// TIA Portal V21 export
FUNCTION_BLOCK "FB104"   // FB104, LAD
TITLE = FB104
{ S7_Optimized_Access := 'FALSE' }
// MANUAL PID
// stored: AutoNumber false, SetENOAutomatically false
   VAR_INPUT
      Enable : Bool;
      SecPulse : Bool;
      AlwaysTrue : Bool;
      DigitalOrAnalog : Bool;   // 0: DIGITAL; 1: ANALOG
      InvertPIDSel : Bool;   // 0: NO; 1: YES
      ActValue : Real;
      SetValue : Real;
      SetPoint1 : Real := 5.0;
      SetPoint2 : Real := 10.0;
      SetPoint3 : Real := 15.0;
      SetPoint4 : Real := 20.0;
      SetPoint5 : Real := 25.0;
      SetPoint6 : Real := 30.0;
      SetPoint7 : Real := 35.0;
      SetPoint8 : Real := 40.0;
      SetPoint9 : Real := 45.0;
      SetPoint10 : Real := 50.0;
      SetRef1 : Real := 10.0;
      SetRef2 : Real := 20.0;
      SetRef3 : Real := 30.0;
      SetRef4 : Real := 40.0;
      SetRef5 : Real := 50.0;
      SetRef6 : Real := 60.0;
      SetRef7 : Real := 70.0;
      SetRef8 : Real := 80.0;
      SetRef9 : Real := 90.0;
      SetRef10 : Real := 100.0;
      OnTime1 : Int := 2;
      OnTime2 : Int := 2;
      OnTime3 : Int := 2;
      OnTime4 : Int := 2;
      OnTime5 : Int := 2;
      OnTime6 : Int := 2;
      OnTime7 : Int := 2;
      OnTime8 : Int := 2;
      OnTime9 : Int := 2;
      OnTime10 : Int := 2;
      OffTime1 : Int := 3;
      OffTime2 : Int := 3;
      OffTime3 : Int := 3;
      OffTime4 : Int := 3;
      OffTime5 : Int := 3;
      OffTime6 : Int := 3;
      OffTime7 : Int := 3;
      OffTime8 : Int := 3;
      OffTime9 : Int := 3;
      OffTime10 : Int := 3;
   END_VAR
   VAR_OUTPUT
      Valve : Bool;
      SetRef : Real;
   END_VAR
   VAR_IN_OUT
      ControlValue1 : Real;
      ControlValue2 : Real;
      ControlValue3 : Real;
      ControlValue4 : Real;
      ControlValue5 : Real;
      ControlValue6 : Real;
      ControlValue7 : Real;
      ControlValue8 : Real;
      ControlValue9 : Real;
      ControlValue10 : Real;
   END_VAR
   VAR
      OnOffDelay { S7_SetPoint := 'True'} : "FB102";
      OnTime : Int;
      OffTime : Int;
   END_VAR
   VAR_TEMP   // added for the SCL form of the ladder/FBD networks
      _w1 : Bool;
   END_VAR
BEGIN

REGION Network 1: Set Point Calculations
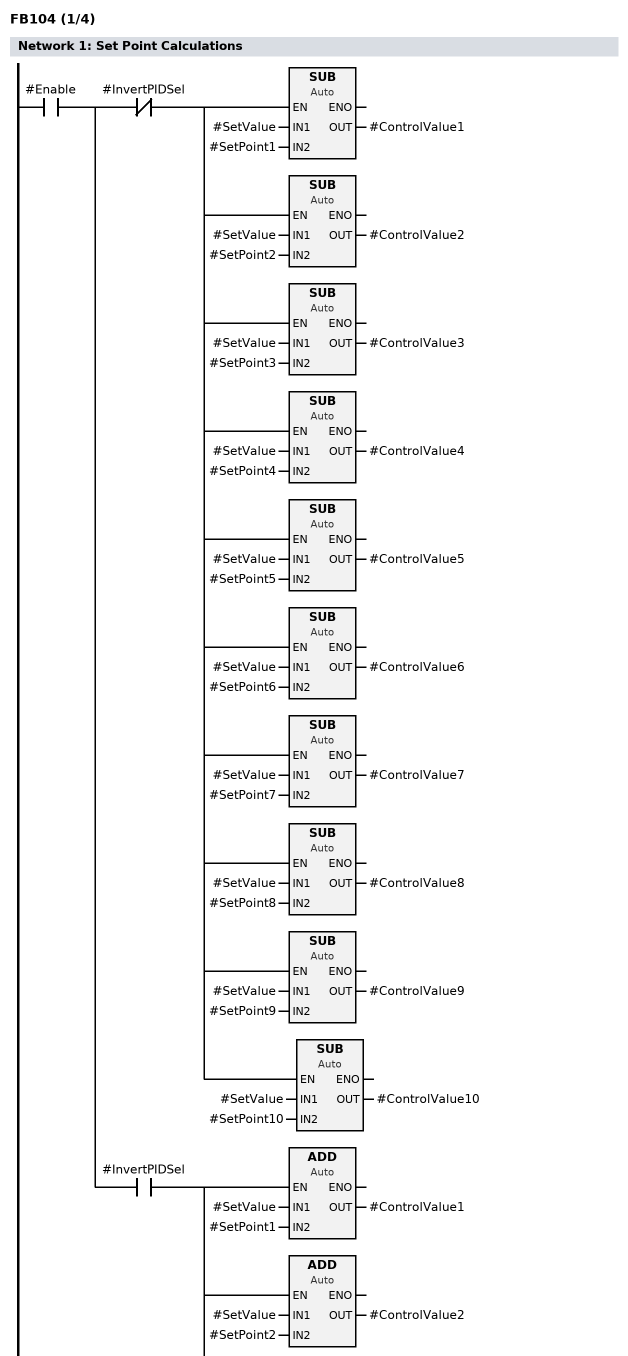
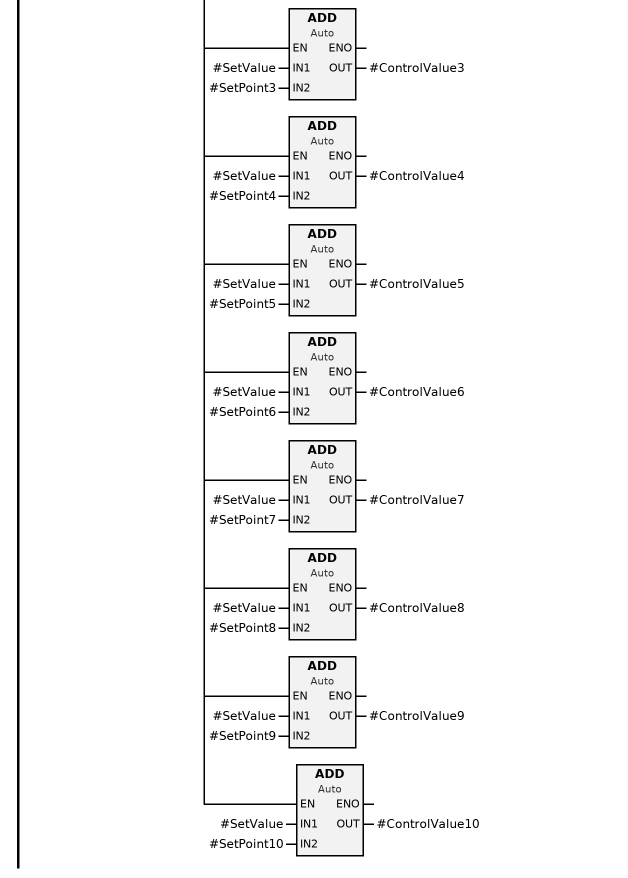
   RUNG wire#powerrail
      Contact( #Enable )
      wire#w1
      I_Contact( #InvertPIDSel )
      wire#w2
      Sub(in1 := #SetValue, in2 := #SetPoint1, out => #ControlValue1)
   END_RUNG
   RUNG wire#w2
      Sub(in1 := #SetValue, in2 := #SetPoint2, out => #ControlValue2)
   END_RUNG
   RUNG wire#w2
      Sub(in1 := #SetValue, in2 := #SetPoint3, out => #ControlValue3)
   END_RUNG
   RUNG wire#w2
      Sub(in1 := #SetValue, in2 := #SetPoint4, out => #ControlValue4)
   END_RUNG
   RUNG wire#w2
      Sub(in1 := #SetValue, in2 := #SetPoint5, out => #ControlValue5)
   END_RUNG
   RUNG wire#w2
      Sub(in1 := #SetValue, in2 := #SetPoint6, out => #ControlValue6)
   END_RUNG
   RUNG wire#w2
      Sub(in1 := #SetValue, in2 := #SetPoint7, out => #ControlValue7)
   END_RUNG
   RUNG wire#w2
      Sub(in1 := #SetValue, in2 := #SetPoint8, out => #ControlValue8)
   END_RUNG
   RUNG wire#w2
      Sub(in1 := #SetValue, in2 := #SetPoint9, out => #ControlValue9)
   END_RUNG
   RUNG wire#w2
      Sub(in1 := #SetValue, in2 := #SetPoint10, out => #ControlValue10)
   END_RUNG
   RUNG wire#w1
      Contact( #InvertPIDSel )
      wire#w3
      Add(in1 := #SetValue, in2 := #SetPoint1, out => #ControlValue1)
   END_RUNG
   RUNG wire#w3
      Add(in1 := #SetValue, in2 := #SetPoint2, out => #ControlValue2)
   END_RUNG
   RUNG wire#w3
      Add(in1 := #SetValue, in2 := #SetPoint3, out => #ControlValue3)
   END_RUNG
   RUNG wire#w3
      Add(in1 := #SetValue, in2 := #SetPoint4, out => #ControlValue4)
   END_RUNG
   RUNG wire#w3
      Add(in1 := #SetValue, in2 := #SetPoint5, out => #ControlValue5)
   END_RUNG
   RUNG wire#w3
      Add(in1 := #SetValue, in2 := #SetPoint6, out => #ControlValue6)
   END_RUNG
   RUNG wire#w3
      Add(in1 := #SetValue, in2 := #SetPoint7, out => #ControlValue7)
   END_RUNG
   RUNG wire#w3
      Add(in1 := #SetValue, in2 := #SetPoint8, out => #ControlValue8)
   END_RUNG
   RUNG wire#w3
      Add(in1 := #SetValue, in2 := #SetPoint9, out => #ControlValue9)
   END_RUNG
   RUNG wire#w3
      Add(in1 := #SetValue, in2 := #SetPoint10, out => #ControlValue10)
   END_RUNG
   // the same network as SCL:
   IF #Enable AND NOT #InvertPIDSel THEN
       #ControlValue1 := #SetValue - #SetPoint1;
       #ControlValue2 := #SetValue - #SetPoint2;
       #ControlValue3 := #SetValue - #SetPoint3;
       #ControlValue4 := #SetValue - #SetPoint4;
       #ControlValue5 := #SetValue - #SetPoint5;
       #ControlValue6 := #SetValue - #SetPoint6;
       #ControlValue7 := #SetValue - #SetPoint7;
       #ControlValue8 := #SetValue - #SetPoint8;
       #ControlValue9 := #SetValue - #SetPoint9;
       #ControlValue10 := #SetValue - #SetPoint10;
   END_IF;
   IF #Enable AND #InvertPIDSel THEN
       #ControlValue1 := #SetValue + #SetPoint1;
       #ControlValue2 := #SetValue + #SetPoint2;
       #ControlValue3 := #SetValue + #SetPoint3;
       #ControlValue4 := #SetValue + #SetPoint4;
       #ControlValue5 := #SetValue + #SetPoint5;
       #ControlValue6 := #SetValue + #SetPoint6;
       #ControlValue7 := #SetValue + #SetPoint7;
       #ControlValue8 := #SetValue + #SetPoint8;
       #ControlValue9 := #SetValue + #SetPoint9;
       #ControlValue10 := #SetValue + #SetPoint10;
   END_IF;
END_REGION

REGION Network 2: Set Reference for InvertPIDSel: NO
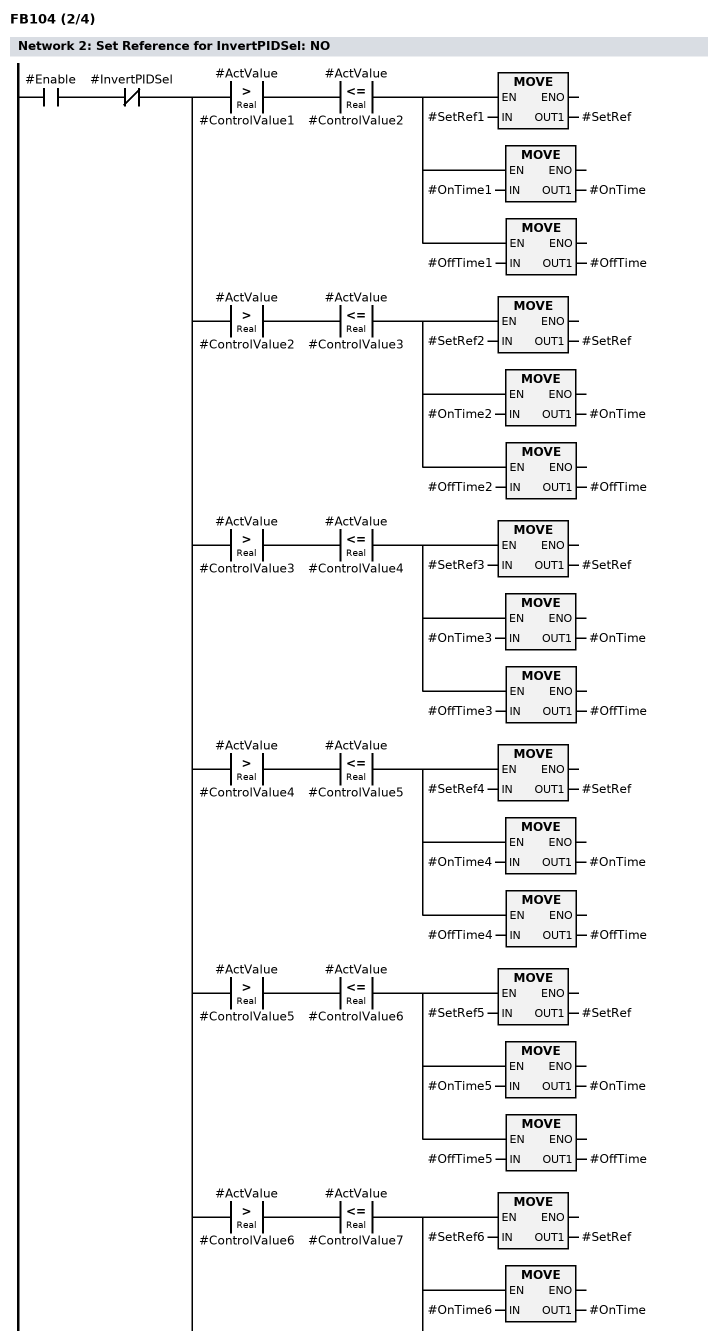
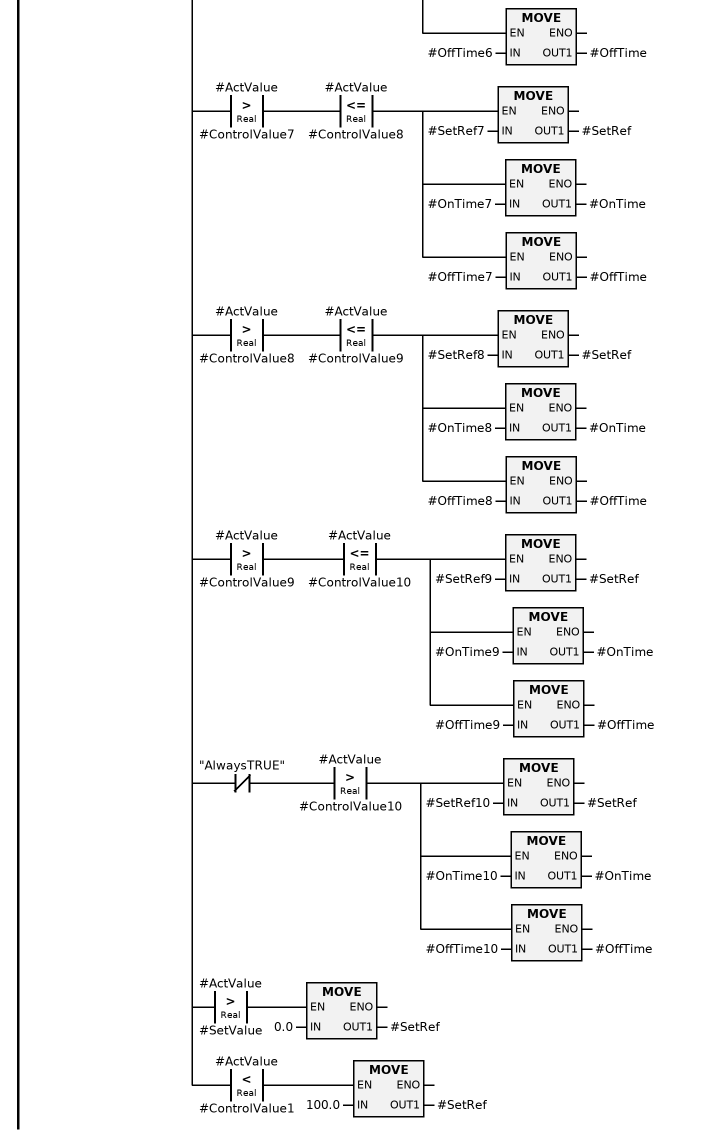
   RUNG wire#powerrail
      Contact( #Enable )
      I_Contact( #InvertPIDSel )
      wire#w1
      { S7_Templates := "SrcType := Real" } GT_Contact(in1 := #ActValue, in2 := #ControlValue1)
      { S7_Templates := "SrcType := Real" } LE_Contact(in1 := #ActValue, in2 := #ControlValue2)
      wire#w2
      Move(in := #SetRef1, out1 => #SetRef)
   END_RUNG
   RUNG wire#w2
      Move(in := #OnTime1, out1 => #OnTime)
   END_RUNG
   RUNG wire#w2
      Move(in := #OffTime1, out1 => #OffTime)
   END_RUNG
   RUNG wire#w1
      { S7_Templates := "SrcType := Real" } GT_Contact(in1 := #ActValue, in2 := #ControlValue2)
      { S7_Templates := "SrcType := Real" } LE_Contact(in1 := #ActValue, in2 := #ControlValue3)
      wire#w3
      Move(in := #SetRef2, out1 => #SetRef)
   END_RUNG
   RUNG wire#w3
      Move(in := #OnTime2, out1 => #OnTime)
   END_RUNG
   RUNG wire#w3
      Move(in := #OffTime2, out1 => #OffTime)
   END_RUNG
   RUNG wire#w1
      { S7_Templates := "SrcType := Real" } GT_Contact(in1 := #ActValue, in2 := #ControlValue3)
      { S7_Templates := "SrcType := Real" } LE_Contact(in1 := #ActValue, in2 := #ControlValue4)
      wire#w4
      Move(in := #SetRef3, out1 => #SetRef)
   END_RUNG
   RUNG wire#w4
      Move(in := #OnTime3, out1 => #OnTime)
   END_RUNG
   RUNG wire#w4
      Move(in := #OffTime3, out1 => #OffTime)
   END_RUNG
   RUNG wire#w1
      { S7_Templates := "SrcType := Real" } GT_Contact(in1 := #ActValue, in2 := #ControlValue4)
      { S7_Templates := "SrcType := Real" } LE_Contact(in1 := #ActValue, in2 := #ControlValue5)
      wire#w5
      Move(in := #SetRef4, out1 => #SetRef)
   END_RUNG
   RUNG wire#w5
      Move(in := #OnTime4, out1 => #OnTime)
   END_RUNG
   RUNG wire#w5
      Move(in := #OffTime4, out1 => #OffTime)
   END_RUNG
   RUNG wire#w1
      { S7_Templates := "SrcType := Real" } GT_Contact(in1 := #ActValue, in2 := #ControlValue5)
      { S7_Templates := "SrcType := Real" } LE_Contact(in1 := #ActValue, in2 := #ControlValue6)
      wire#w6
      Move(in := #SetRef5, out1 => #SetRef)
   END_RUNG
   RUNG wire#w6
      Move(in := #OnTime5, out1 => #OnTime)
   END_RUNG
   RUNG wire#w6
      Move(in := #OffTime5, out1 => #OffTime)
   END_RUNG
   RUNG wire#w1
      { S7_Templates := "SrcType := Real" } GT_Contact(in1 := #ActValue, in2 := #ControlValue6)
      { S7_Templates := "SrcType := Real" } LE_Contact(in1 := #ActValue, in2 := #ControlValue7)
      wire#w7
      Move(in := #SetRef6, out1 => #SetRef)
   END_RUNG
   RUNG wire#w7
      Move(in := #OnTime6, out1 => #OnTime)
   END_RUNG
   RUNG wire#w7
      Move(in := #OffTime6, out1 => #OffTime)
   END_RUNG
   RUNG wire#w1
      { S7_Templates := "SrcType := Real" } GT_Contact(in1 := #ActValue, in2 := #ControlValue7)
      { S7_Templates := "SrcType := Real" } LE_Contact(in1 := #ActValue, in2 := #ControlValue8)
      wire#w8
      Move(in := #SetRef7, out1 => #SetRef)
   END_RUNG
   RUNG wire#w8
      Move(in := #OnTime7, out1 => #OnTime)
   END_RUNG
   RUNG wire#w8
      Move(in := #OffTime7, out1 => #OffTime)
   END_RUNG
   RUNG wire#w1
      { S7_Templates := "SrcType := Real" } GT_Contact(in1 := #ActValue, in2 := #ControlValue8)
      { S7_Templates := "SrcType := Real" } LE_Contact(in1 := #ActValue, in2 := #ControlValue9)
      wire#w9
      Move(in := #SetRef8, out1 => #SetRef)
   END_RUNG
   RUNG wire#w9
      Move(in := #OnTime8, out1 => #OnTime)
   END_RUNG
   RUNG wire#w9
      Move(in := #OffTime8, out1 => #OffTime)
   END_RUNG
   RUNG wire#w1
      { S7_Templates := "SrcType := Real" } GT_Contact(in1 := #ActValue, in2 := #ControlValue9)
      { S7_Templates := "SrcType := Real" } LE_Contact(in1 := #ActValue, in2 := #ControlValue10)
      wire#w10
      Move(in := #SetRef9, out1 => #SetRef)
   END_RUNG
   RUNG wire#w10
      Move(in := #OnTime9, out1 => #OnTime)
   END_RUNG
   RUNG wire#w10
      Move(in := #OffTime9, out1 => #OffTime)
   END_RUNG
   RUNG wire#w1
      I_Contact( "AlwaysTRUE" )
      { S7_Templates := "SrcType := Real" } GT_Contact(in1 := #ActValue, in2 := #ControlValue10)
      wire#w11
      Move(in := #SetRef10, out1 => #SetRef)
   END_RUNG
   RUNG wire#w11
      Move(in := #OnTime10, out1 => #OnTime)
   END_RUNG
   RUNG wire#w11
      Move(in := #OffTime10, out1 => #OffTime)
   END_RUNG
   RUNG wire#w1
      { S7_Templates := "SrcType := Real" } GT_Contact(in1 := #ActValue, in2 := #SetValue)
      Move(in := 0.0, out1 => #SetRef)
   END_RUNG
   RUNG wire#w1
      { S7_Templates := "SrcType := Real" } LT_Contact(in1 := #ActValue, in2 := #ControlValue1)
      Move(in := 100.0, out1 => #SetRef)
   END_RUNG
   // the same network as SCL:
   #_w1 := #Enable AND NOT #InvertPIDSel;
   IF #_w1 AND (#ActValue > #ControlValue1) AND (#ActValue <= #ControlValue2) THEN
       #SetRef := #SetRef1;
       #OnTime := #OnTime1;
       #OffTime := #OffTime1;
   END_IF;
   IF #_w1 AND (#ActValue > #ControlValue2) AND (#ActValue <= #ControlValue3) THEN
       #SetRef := #SetRef2;
       #OnTime := #OnTime2;
       #OffTime := #OffTime2;
   END_IF;
   IF #_w1 AND (#ActValue > #ControlValue3) AND (#ActValue <= #ControlValue4) THEN
       #SetRef := #SetRef3;
       #OnTime := #OnTime3;
       #OffTime := #OffTime3;
   END_IF;
   IF #_w1 AND (#ActValue > #ControlValue4) AND (#ActValue <= #ControlValue5) THEN
       #SetRef := #SetRef4;
       #OnTime := #OnTime4;
       #OffTime := #OffTime4;
   END_IF;
   IF #_w1 AND (#ActValue > #ControlValue5) AND (#ActValue <= #ControlValue6) THEN
       #SetRef := #SetRef5;
       #OnTime := #OnTime5;
       #OffTime := #OffTime5;
   END_IF;
   IF #_w1 AND (#ActValue > #ControlValue6) AND (#ActValue <= #ControlValue7) THEN
       #SetRef := #SetRef6;
       #OnTime := #OnTime6;
       #OffTime := #OffTime6;
   END_IF;
   IF #_w1 AND (#ActValue > #ControlValue7) AND (#ActValue <= #ControlValue8) THEN
       #SetRef := #SetRef7;
       #OnTime := #OnTime7;
       #OffTime := #OffTime7;
   END_IF;
   IF #_w1 AND (#ActValue > #ControlValue8) AND (#ActValue <= #ControlValue9) THEN
       #SetRef := #SetRef8;
       #OnTime := #OnTime8;
       #OffTime := #OffTime8;
   END_IF;
   IF #_w1 AND (#ActValue > #ControlValue9) AND (#ActValue <= #ControlValue10) THEN
       #SetRef := #SetRef9;
       #OnTime := #OnTime9;
       #OffTime := #OffTime9;
   END_IF;
   IF #_w1 AND NOT "AlwaysTRUE" AND (#ActValue > #ControlValue10) THEN
       #SetRef := #SetRef10;
       #OnTime := #OnTime10;
       #OffTime := #OffTime10;
   END_IF;
   IF #_w1 AND (#ActValue > #SetValue) THEN #SetRef := 0.0; END_IF;
   IF #_w1 AND (#ActValue < #ControlValue1) THEN #SetRef := 100.0; END_IF;
END_REGION

REGION Network 3: Set Reference for InvertPIDSel: YES
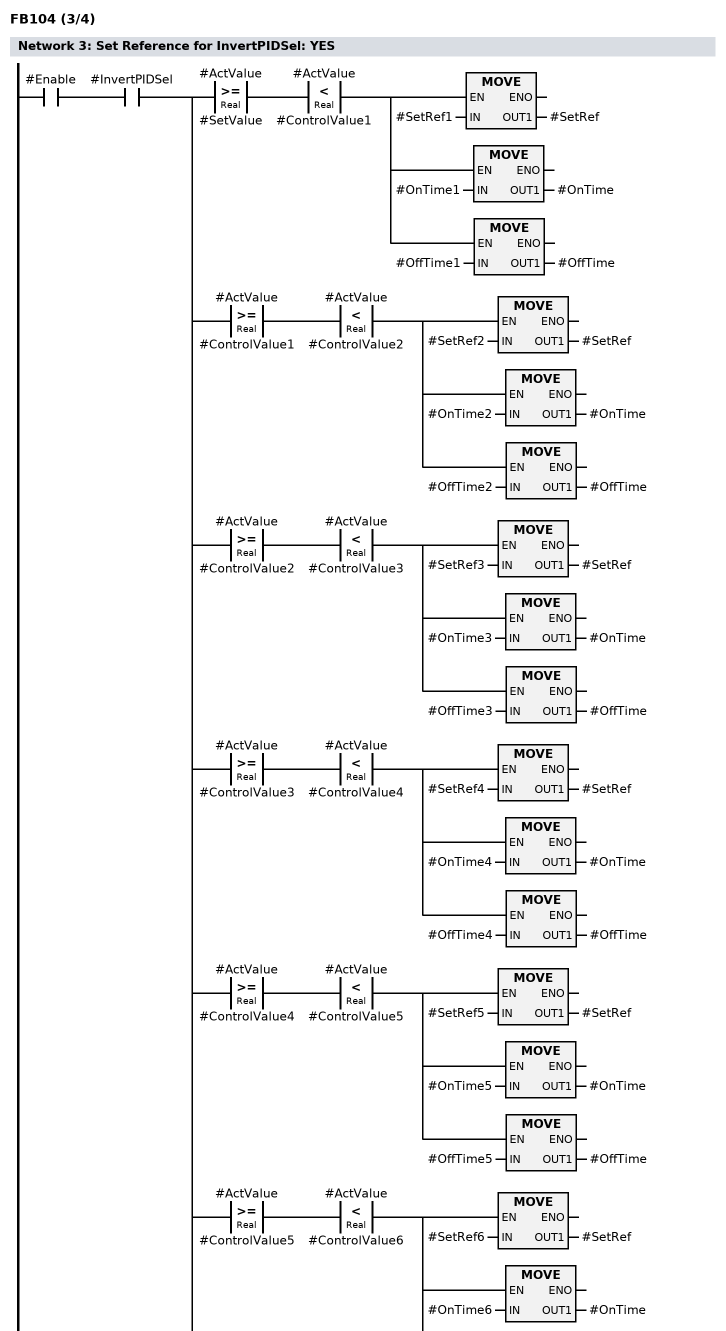
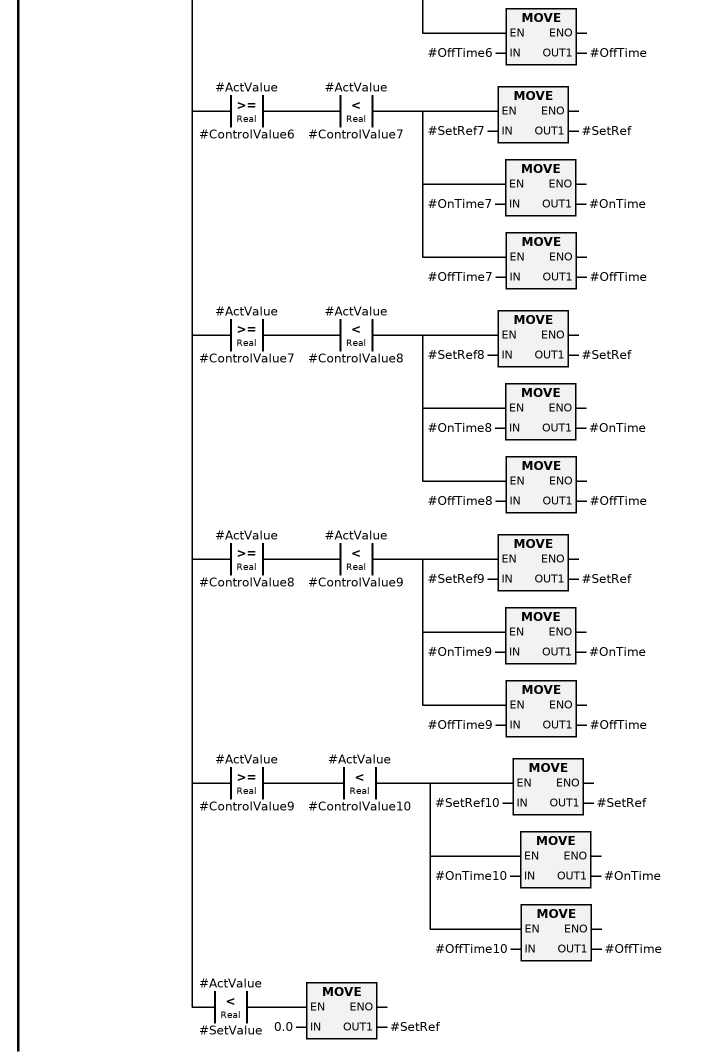
   RUNG wire#powerrail
      Contact( #Enable )
      Contact( #InvertPIDSel )
      wire#w1
      { S7_Templates := "SrcType := Real" } GE_Contact(in1 := #ActValue, in2 := #SetValue)
      { S7_Templates := "SrcType := Real" } LT_Contact(in1 := #ActValue, in2 := #ControlValue1)
      wire#w2
      Move(in := #SetRef1, out1 => #SetRef)
   END_RUNG
   RUNG wire#w2
      Move(in := #OnTime1, out1 => #OnTime)
   END_RUNG
   RUNG wire#w2
      Move(in := #OffTime1, out1 => #OffTime)
   END_RUNG
   RUNG wire#w1
      { S7_Templates := "SrcType := Real" } GE_Contact(in1 := #ActValue, in2 := #ControlValue1)
      { S7_Templates := "SrcType := Real" } LT_Contact(in1 := #ActValue, in2 := #ControlValue2)
      wire#w3
      Move(in := #SetRef2, out1 => #SetRef)
   END_RUNG
   RUNG wire#w3
      Move(in := #OnTime2, out1 => #OnTime)
   END_RUNG
   RUNG wire#w3
      Move(in := #OffTime2, out1 => #OffTime)
   END_RUNG
   RUNG wire#w1
      { S7_Templates := "SrcType := Real" } GE_Contact(in1 := #ActValue, in2 := #ControlValue2)
      { S7_Templates := "SrcType := Real" } LT_Contact(in1 := #ActValue, in2 := #ControlValue3)
      wire#w4
      Move(in := #SetRef3, out1 => #SetRef)
   END_RUNG
   RUNG wire#w4
      Move(in := #OnTime3, out1 => #OnTime)
   END_RUNG
   RUNG wire#w4
      Move(in := #OffTime3, out1 => #OffTime)
   END_RUNG
   RUNG wire#w1
      { S7_Templates := "SrcType := Real" } GE_Contact(in1 := #ActValue, in2 := #ControlValue3)
      { S7_Templates := "SrcType := Real" } LT_Contact(in1 := #ActValue, in2 := #ControlValue4)
      wire#w5
      Move(in := #SetRef4, out1 => #SetRef)
   END_RUNG
   RUNG wire#w5
      Move(in := #OnTime4, out1 => #OnTime)
   END_RUNG
   RUNG wire#w5
      Move(in := #OffTime4, out1 => #OffTime)
   END_RUNG
   RUNG wire#w1
      { S7_Templates := "SrcType := Real" } GE_Contact(in1 := #ActValue, in2 := #ControlValue4)
      { S7_Templates := "SrcType := Real" } LT_Contact(in1 := #ActValue, in2 := #ControlValue5)
      wire#w6
      Move(in := #SetRef5, out1 => #SetRef)
   END_RUNG
   RUNG wire#w6
      Move(in := #OnTime5, out1 => #OnTime)
   END_RUNG
   RUNG wire#w6
      Move(in := #OffTime5, out1 => #OffTime)
   END_RUNG
   RUNG wire#w1
      { S7_Templates := "SrcType := Real" } GE_Contact(in1 := #ActValue, in2 := #ControlValue5)
      { S7_Templates := "SrcType := Real" } LT_Contact(in1 := #ActValue, in2 := #ControlValue6)
      wire#w7
      Move(in := #SetRef6, out1 => #SetRef)
   END_RUNG
   RUNG wire#w7
      Move(in := #OnTime6, out1 => #OnTime)
   END_RUNG
   RUNG wire#w7
      Move(in := #OffTime6, out1 => #OffTime)
   END_RUNG
   RUNG wire#w1
      { S7_Templates := "SrcType := Real" } GE_Contact(in1 := #ActValue, in2 := #ControlValue6)
      { S7_Templates := "SrcType := Real" } LT_Contact(in1 := #ActValue, in2 := #ControlValue7)
      wire#w8
      Move(in := #SetRef7, out1 => #SetRef)
   END_RUNG
   RUNG wire#w8
      Move(in := #OnTime7, out1 => #OnTime)
   END_RUNG
   RUNG wire#w8
      Move(in := #OffTime7, out1 => #OffTime)
   END_RUNG
   RUNG wire#w1
      { S7_Templates := "SrcType := Real" } GE_Contact(in1 := #ActValue, in2 := #ControlValue7)
      { S7_Templates := "SrcType := Real" } LT_Contact(in1 := #ActValue, in2 := #ControlValue8)
      wire#w9
      Move(in := #SetRef8, out1 => #SetRef)
   END_RUNG
   RUNG wire#w9
      Move(in := #OnTime8, out1 => #OnTime)
   END_RUNG
   RUNG wire#w9
      Move(in := #OffTime8, out1 => #OffTime)
   END_RUNG
   RUNG wire#w1
      { S7_Templates := "SrcType := Real" } GE_Contact(in1 := #ActValue, in2 := #ControlValue8)
      { S7_Templates := "SrcType := Real" } LT_Contact(in1 := #ActValue, in2 := #ControlValue9)
      wire#w10
      Move(in := #SetRef9, out1 => #SetRef)
   END_RUNG
   RUNG wire#w10
      Move(in := #OnTime9, out1 => #OnTime)
   END_RUNG
   RUNG wire#w10
      Move(in := #OffTime9, out1 => #OffTime)
   END_RUNG
   RUNG wire#w1
      { S7_Templates := "SrcType := Real" } GE_Contact(in1 := #ActValue, in2 := #ControlValue9)
      { S7_Templates := "SrcType := Real" } LT_Contact(in1 := #ActValue, in2 := #ControlValue10)
      wire#w11
      Move(in := #SetRef10, out1 => #SetRef)
   END_RUNG
   RUNG wire#w11
      Move(in := #OnTime10, out1 => #OnTime)
   END_RUNG
   RUNG wire#w11
      Move(in := #OffTime10, out1 => #OffTime)
   END_RUNG
   RUNG wire#w1
      { S7_Templates := "SrcType := Real" } LT_Contact(in1 := #ActValue, in2 := #SetValue)
      Move(in := 0.0, out1 => #SetRef)
   END_RUNG
   // the same network as SCL:
   #_w1 := #Enable AND #InvertPIDSel;
   IF #_w1 AND (#ActValue >= #SetValue) AND (#ActValue < #ControlValue1) THEN
       #SetRef := #SetRef1;
       #OnTime := #OnTime1;
       #OffTime := #OffTime1;
   END_IF;
   IF #_w1 AND (#ActValue >= #ControlValue1) AND (#ActValue < #ControlValue2) THEN
       #SetRef := #SetRef2;
       #OnTime := #OnTime2;
       #OffTime := #OffTime2;
   END_IF;
   IF #_w1 AND (#ActValue >= #ControlValue2) AND (#ActValue < #ControlValue3) THEN
       #SetRef := #SetRef3;
       #OnTime := #OnTime3;
       #OffTime := #OffTime3;
   END_IF;
   IF #_w1 AND (#ActValue >= #ControlValue3) AND (#ActValue < #ControlValue4) THEN
       #SetRef := #SetRef4;
       #OnTime := #OnTime4;
       #OffTime := #OffTime4;
   END_IF;
   IF #_w1 AND (#ActValue >= #ControlValue4) AND (#ActValue < #ControlValue5) THEN
       #SetRef := #SetRef5;
       #OnTime := #OnTime5;
       #OffTime := #OffTime5;
   END_IF;
   IF #_w1 AND (#ActValue >= #ControlValue5) AND (#ActValue < #ControlValue6) THEN
       #SetRef := #SetRef6;
       #OnTime := #OnTime6;
       #OffTime := #OffTime6;
   END_IF;
   IF #_w1 AND (#ActValue >= #ControlValue6) AND (#ActValue < #ControlValue7) THEN
       #SetRef := #SetRef7;
       #OnTime := #OnTime7;
       #OffTime := #OffTime7;
   END_IF;
   IF #_w1 AND (#ActValue >= #ControlValue7) AND (#ActValue < #ControlValue8) THEN
       #SetRef := #SetRef8;
       #OnTime := #OnTime8;
       #OffTime := #OffTime8;
   END_IF;
   IF #_w1 AND (#ActValue >= #ControlValue8) AND (#ActValue < #ControlValue9) THEN
       #SetRef := #SetRef9;
       #OnTime := #OnTime9;
       #OffTime := #OffTime9;
   END_IF;
   IF #_w1 AND (#ActValue >= #ControlValue9) AND (#ActValue < #ControlValue10) THEN
       #SetRef := #SetRef10;
       #OnTime := #OnTime10;
       #OffTime := #OffTime10;
   END_IF;
   IF #_w1 AND (#ActValue < #SetValue) THEN #SetRef := 0.0; END_IF;
END_REGION

REGION Network 4: On/Off Delay
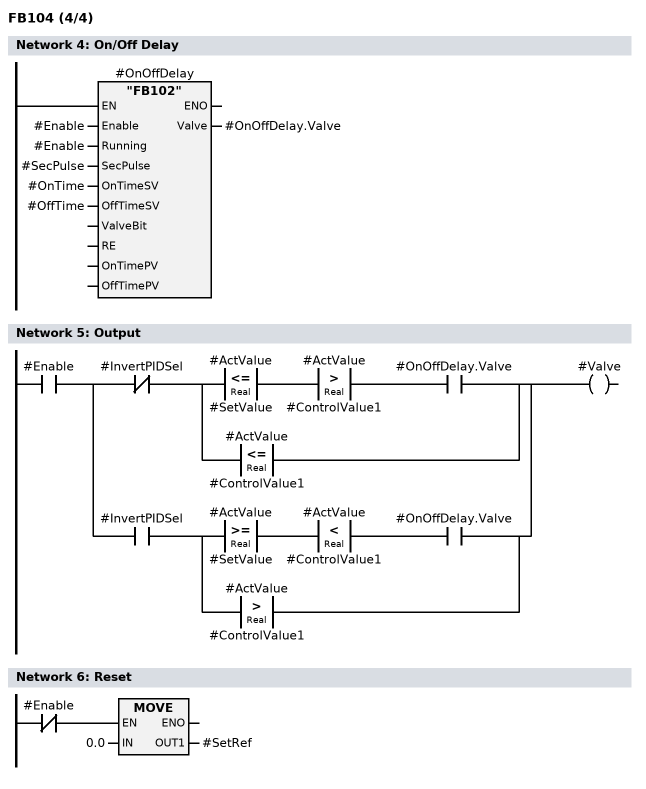
   RUNG wire#powerrail
      #OnOffDelay(Enable := #Enable, Running := #Enable, SecPulse := #SecPulse, OnTimeSV := #OnTime, OffTimeSV := #OffTime, ValveBit :=, RE :=, OnTimePV :=, OffTimePV :=, Valve => #OnOffDelay.Valve)
   END_RUNG
   // the same network as SCL:
   #OnOffDelay(Enable := #Enable,   // "FB102"
               Running := #Enable,
               SecPulse := #SecPulse,
               OnTimeSV := #OnTime,
               OffTimeSV := #OffTime,
               Valve => #OnOffDelay.Valve);
END_REGION

REGION Network 5: Output
   RUNG wire#powerrail
      Contact( #Enable )
      wire#w1
      I_Contact( #InvertPIDSel )
      wire#w2
      { S7_Templates := "SrcType := Real" } LE_Contact(in1 := #ActValue, in2 := #SetValue)
      { S7_Templates := "SrcType := Real" } GT_Contact(in1 := #ActValue, in2 := #ControlValue1)
      Contact( #OnOffDelay.Valve )
      wire#w3
      Coil( #Valve )
   END_RUNG
   RUNG wire#w2
      { S7_Templates := "SrcType := Real" } LE_Contact(in1 := #ActValue, in2 := #ControlValue1)
   END_RUNG wire#w3
   RUNG wire#w1
      Contact( #InvertPIDSel )
      wire#w4
      { S7_Templates := "SrcType := Real" } GE_Contact(in1 := #ActValue, in2 := #SetValue)
      { S7_Templates := "SrcType := Real" } LT_Contact(in1 := #ActValue, in2 := #ControlValue1)
      Contact( #OnOffDelay.Valve )
   END_RUNG wire#w3
   RUNG wire#w4
      { S7_Templates := "SrcType := Real" } GT_Contact(in1 := #ActValue, in2 := #ControlValue1)
   END_RUNG wire#w3
   // the same network as SCL:
   #Valve := #Enable AND ((NOT #InvertPIDSel AND (((#ActValue <= #SetValue) AND (#ActValue > #ControlValue1) AND #OnOffDelay.Valve) OR (#ActValue <= #ControlValue1))) OR (#InvertPIDSel AND (((#ActValue >= #SetValue) AND (#ActValue < #ControlValue1) AND #OnOffDelay.Valve) OR (#ActValue > #ControlValue1))));
END_REGION

REGION Network 6: Reset
   RUNG wire#powerrail
      I_Contact( #Enable )
      Move(in := 0.0, out1 => #SetRef)
   END_RUNG
   // the same network as SCL:
   IF NOT #Enable THEN #SetRef := 0.0; END_IF;
END_REGION
END_FUNCTION_BLOCK
